INTERFACE I_Parameters

METHOD PUBLIC Accept
VAR_INPUT
	Visitor : I_ParameterVisitor;
END_VAR
END_METHOD

METHOD PUBLIC AddDataAsParameter : I_Parameter
VAR_INPUT
	Name : T_MAXSTRING;
	Data : I_Datatype;
END_VAR
END_METHOD

METHOD AddParameter
VAR_INPUT
	Parameter : I_Parameter;
END_VAR
END_METHOD

METHOD PUBLIC TryGetParameterByName : BOOL
VAR_INPUT
	Name : T_MAXSTRING;
	Destination : REFERENCE TO I_Parameter;
END_VAR
END_METHOD

END_INTERFACE

(* stored: Version 1.1.0.1, ProductVersion 3.1.4024.12
   Itf I_Parameters: Id {062edb1f-457b-4873-87d5-c259f2c488a1}
   Method Accept: Id {3a16eb56-84de-4cbe-93df-840b6a1e6e37}
   Method AddDataAsParameter: Id {19236629-dcdf-4757-afa1-0f5ce88c51e2}
   Method AddParameter: Id {0a3fa470-91f6-4109-be0b-6b4f3fdd3712}
   Method TryGetParameterByName: Id {69d9d93c-b35b-43f3-a3f1-7dfd1697741f} *)
